FUNCTION_BLOCK FB_FlowCalcs
VAR_INPUT
END_VAR
VAR_OUTPUT
END_VAR
VAR
END_VAR

END_FUNCTION_BLOCK

(* stored: Version 1.1.0.1, ProductVersion 3.1.4026.18
   POU FB_FlowCalcs: Id {1756219a-0231-4cbf-99e3-e5ecc1f6178b}, SpecialFunc None *)
